Staubli VAL3: AXISMOVER.pjx

--- AXISMOVER.pjx ---
Parameters version=s7.2.1 stackSize=5000 millimeterUnit=true
Program file=find.pgx
Program file=get.pgx
Program file=getSize.pgx
Program file=loadCycle.pgx
Program file=onEdit.pgx
Program file=onInsert.pgx
Program file=onProgEnd.pgx
Program file=onRun.pgx
Program file=onStart.pgx
Program file=onStop.pgx
Data file=AXISMOVER.dtx
Library alias=io path=Disk://io/io.pjx
Library alias=use path=Disk://kernel/userPage/userPage.pjx

--- AXISMOVER.dtx ---
public string sItems
public bool bAxisMove

--- get.pgx ---
public program get(string& x_sItem[], num x_nIndex)
begin
end

--- onEdit.pgx ---
public program onEdit(string& x_sItem[])
  local num l_nX
  local num l_nY
  local num l_nDelay
begin
  // convert to a num
  toNum(x_sItem,l_nDelay,true)
  // change the field
  call use:insertDialog("Distance [mm] ",l_nDelay,-0.01,2680.01)
  // give back
  if l_nDelay>=0
    l_nDelay=round(l_nDelay)
    x_sItem="AXISMOVER "+toString("",l_nDelay)
  endIf
end

--- onInsert.pgx ---
public program onInsert(string& x_sItem[])
  local num l_nDelay
begin
  cls()
  l_nDelay=0
  call use:insertDialog("Distance [mm] ",l_nDelay,-0.01,2680.01)
  // give back
  if l_nDelay>=0
    l_nDelay=round(l_nDelay)
    x_sItem="AXISMOVER "+toString("",l_nDelay)
  endIf
end

--- onRun.pgx ---
public program onRun(string& x_sItem[])
  local num l_nValue
  local num l_nVelocity
begin
  //
  // convert to a num

  bAxisMove=true
  aioSet(io:MbAO_b8Axis,1)
  aioSet(io:MbAO_bMoveToPos,0)
  toNum(x_sItem,l_nValue,true)
  // NB the robot will no STOP
//  aioSet(io:MbAI_bAxis8Reac,0)
  delay(0.5)
  l_nVelocity=speedScale()
  l_nVelocity=700*l_nVelocity/100
  l_nVelocity=round(l_nVelocity)
  l_nValue=round(l_nValue)
  aioSet(io:MbAO_aMovePosL8,0)
  aioSet(io:MbAO_aMovePosH8,2.554265*l_nValue)
  aioSet(io:MbAO_aMoveDis8,1)
  aioSet(io:MbAO_aVelocity8,l_nVelocity)
  aioSet(io:MbAO_bMovePos8,1)
  delay(0.5)
  wait(aioGet(io:MbAI_bAxis8Reac)==0)
  wait(aioGet(io:MbAI_bAxis8Reac)==1)
  aioSet(io:MbAO_bMovePos8,0)
  aioSet(io:MbAO_aMoveDis8,0)
  aioSet(io:MbAO_b8Axis,0)
  bAxisMove=false
end

--- onStart.pgx ---
public program onStart(string& x_sItem[])
begin
end

--- onStop.pgx ---
public program onStop(string& x_sItem[])
begin
  aioSet(io:MbAO_aMoveDis,0)
  //aioSet(io:MbAO_b7Axis,0)
  //logMsg("8")
end
